PROGRAM F12_PackerQueuesCtrl
VAR

	rtrigScanBarcode				: R_TRIG;
	fbScannerCtrl					: FB_SCANNER_CameraSelect;
	fbImageBuffer					: FB_CASE_LastRowPoisitionBuffer_v2;
	fbCaseContentEvaluation			: FB_SCANNER_Evaluation;

	bShiftBufferDone						: BOOL;

	ctuAuxRowCounter				: CTU;
	nAuxRowIndex						: INT;
	rtrigAuxRowComplete				: R_TRIG;	(*option*)

	fbCaseInspectionSeq			: FB_SYSTEM_SeqControl;
	nSequenceStep				: INT;
	b00_Idle						: BOOL;
	b01_ScanBarcode				: BOOL;
	b06_MoveOutersToCaseData		: BOOL;
	b20_Done						: BOOL;

	bBusy						: BOOL;
	fbScanTimeout					: TON;

	fbFailedReadCounter			: CTU;
	fbMoveOuterToCaseDataPosition	: FB_CASE_MoveOutersRowToPacker;
	rtrigCaseContentValidation				: R_TRIG;

	fbValidationIndexOK						: FB_CTU32;
	fbValidationIndexUnder					: FB_CTU32;
	fbValidationIndexOver					: FB_CTU32;
	fbValidationNotFound					: FB_CTU32;

	tofCaseContentCameraOFFDelay 	: TOF;
	bTest	: BOOL;


	fbDebugCNT				: FB_DEBUG_CounterArray;
	aCNTDebug				: ARRAY [1..10] OF UDINT;
	bResetCNT					: BOOL;

END_VAR
(*
VAR CONSTANT
	sOptions						: ST_SCANNER_Options := (eScannerType := E_MV_420_FULL, nImageBuffer := 1, nExpectedResp := 1);
END_VAR*)

(*
Modification history:
Date		|	Author 		|	Remark
----------------------------------------------------------------------------------------------------
02.09.20	|	PP			|	Start Remarking.
*)
VAR // added by the converter: edge detectors and wires of the graphical bodies
    _w1 : BOOL;
END_VAR

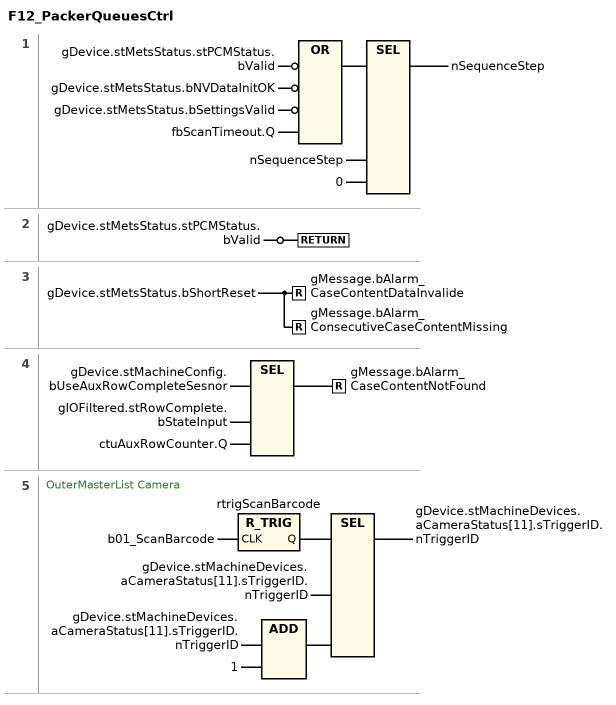
// NETWORK 1
nSequenceStep := SEL(NOT gDevice.stMetsStatus.stPCMStatus.bValid OR NOT gDevice.stMetsStatus.bNVDataInitOK OR NOT gDevice.stMetsStatus.bSettingsValid OR fbScanTimeout.Q, nSequenceStep, 0);

// NETWORK 2
IF NOT gDevice.stMetsStatus.stPCMStatus.bValid THEN RETURN; END_IF

// NETWORK 3
gMessage.bAlarm_CaseContentDataInvalide R= gDevice.stMetsStatus.bShortReset;
gMessage.bAlarm_ConsecutiveCaseContentMissing R= gDevice.stMetsStatus.bShortReset;

// NETWORK 4
gMessage.bAlarm_CaseContentNotFound R= SEL(gDevice.stMachineConfig.bUseAuxRowCompleteSesnor, gIOFiltered.stRowComplete.bStateInput, ctuAuxRowCounter.Q);

// NETWORK 5
// OuterMasterList Camera
rtrigScanBarcode(CLK := b01_ScanBarcode); // R_TRIG
gDevice.stMachineDevices.aCameraStatus[11].sTriggerID.nTriggerID := SEL(rtrigScanBarcode.Q, gDevice.stMachineDevices.aCameraStatus[11].sTriggerID.nTriggerID, gDevice.stMachineDevices.aCameraStatus[11].sTriggerID.nTriggerID + 1);

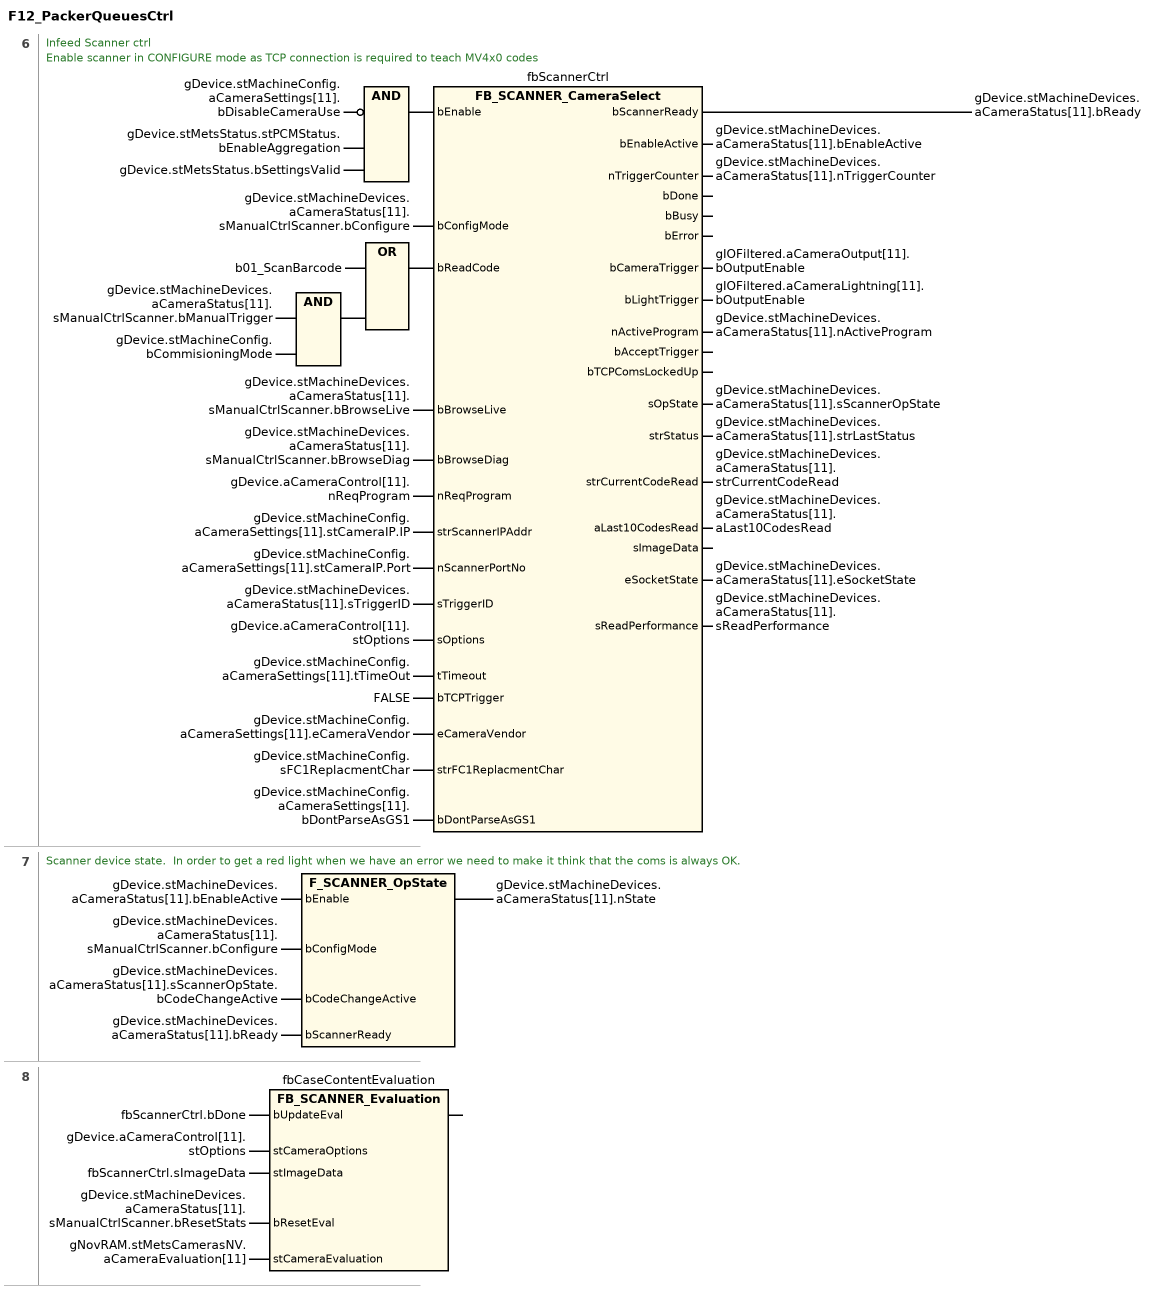
// NETWORK 6
// 					Infeed Scanner ctrl
// Enable scanner in CONFIGURE mode as TCP connection is required to teach MV4x0 codes
//
fbScannerCtrl(
    bEnable := NOT gDevice.stMachineConfig.aCameraSettings[11].bDisableCameraUse AND gDevice.stMetsStatus.stPCMStatus.bEnableAggregation AND gDevice.stMetsStatus.bSettingsValid,
    bConfigMode := gDevice.stMachineDevices.aCameraStatus[11].sManualCtrlScanner.bConfigure,
    bReadCode := b01_ScanBarcode OR gDevice.stMachineDevices.aCameraStatus[11].sManualCtrlScanner.bManualTrigger AND gDevice.stMachineConfig.bCommisioningMode,
    bBrowseLive := gDevice.stMachineDevices.aCameraStatus[11].sManualCtrlScanner.bBrowseLive,
    bBrowseDiag := gDevice.stMachineDevices.aCameraStatus[11].sManualCtrlScanner.bBrowseDiag,
    nReqProgram := gDevice.aCameraControl[11].nReqProgram,
    strScannerIPAddr := gDevice.stMachineConfig.aCameraSettings[11].stCameraIP.IP,
    nScannerPortNo := gDevice.stMachineConfig.aCameraSettings[11].stCameraIP.Port,
    sTriggerID := gDevice.stMachineDevices.aCameraStatus[11].sTriggerID,
    sOptions := gDevice.aCameraControl[11].stOptions,
    tTimeout := gDevice.stMachineConfig.aCameraSettings[11].tTimeOut,
    bTCPTrigger := FALSE,
    eCameraVendor := gDevice.stMachineConfig.aCameraSettings[11].eCameraVendor,
    strFC1ReplacmentChar := gDevice.stMachineConfig.sFC1ReplacmentChar,
    bDontParseAsGS1 := gDevice.stMachineConfig.aCameraSettings[11].bDontParseAsGS1,
    bEnableActive => gDevice.stMachineDevices.aCameraStatus[11].bEnableActive,
    nTriggerCounter => gDevice.stMachineDevices.aCameraStatus[11].nTriggerCounter,
    bCameraTrigger => gIOFiltered.aCameraOutput[11].bOutputEnable,
    bLightTrigger => gIOFiltered.aCameraLightning[11].bOutputEnable,
    nActiveProgram => gDevice.stMachineDevices.aCameraStatus[11].nActiveProgram,
    sOpState => gDevice.stMachineDevices.aCameraStatus[11].sScannerOpState,
    strStatus => gDevice.stMachineDevices.aCameraStatus[11].strLastStatus,
    strCurrentCodeRead => gDevice.stMachineDevices.aCameraStatus[11].strCurrentCodeRead,
    aLast10CodesRead => gDevice.stMachineDevices.aCameraStatus[11].aLast10CodesRead,
    eSocketState => gDevice.stMachineDevices.aCameraStatus[11].eSocketState,
    sReadPerformance => gDevice.stMachineDevices.aCameraStatus[11].sReadPerformance); // FB_SCANNER_CameraSelect
gDevice.stMachineDevices.aCameraStatus[11].bReady := fbScannerCtrl.bScannerReady;

// NETWORK 7
// Scanner device state.  In order to get a red light when we have an error we need to make it think that the coms is always OK.
gDevice.stMachineDevices.aCameraStatus[11].nState := F_SCANNER_OpState(bEnable := gDevice.stMachineDevices.aCameraStatus[11].bEnableActive, bConfigMode := gDevice.stMachineDevices.aCameraStatus[11].sManualCtrlScanner.bConfigure, bCodeChangeActive := gDevice.stMachineDevices.aCameraStatus[11].sScannerOpState.bCodeChangeActive, bScannerReady := gDevice.stMachineDevices.aCameraStatus[11].bReady);

// NETWORK 8
fbCaseContentEvaluation(
    bUpdateEval := fbScannerCtrl.bDone,
    stCameraOptions := gDevice.aCameraControl[11].stOptions,
    stImageData := fbScannerCtrl.sImageData,
    bResetEval := gDevice.stMachineDevices.aCameraStatus[11].sManualCtrlScanner.bResetStats,
    stCameraEvaluation := gNovRAM.stMetsCamerasNV.aCameraEvaluation[11]); // FB_SCANNER_Evaluation

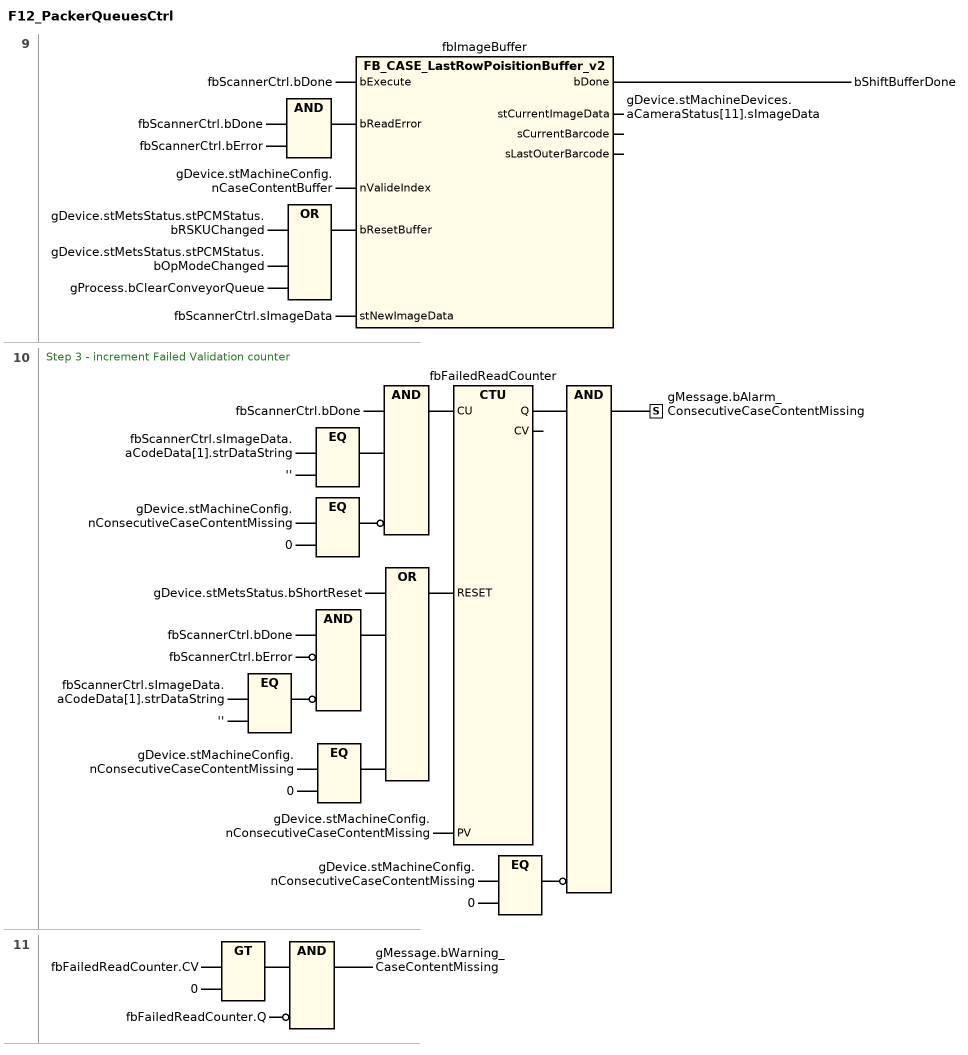
// NETWORK 9
fbImageBuffer(
    bExecute := fbScannerCtrl.bDone,
    bReadError := fbScannerCtrl.bDone AND fbScannerCtrl.bError,
    nValideIndex := gDevice.stMachineConfig.nCaseContentBuffer,
    bResetBuffer := gDevice.stMetsStatus.stPCMStatus.bRSKUChanged OR gDevice.stMetsStatus.stPCMStatus.bOpModeChanged OR gProcess.bClearConveyorQueue,
    stNewImageData := fbScannerCtrl.sImageData,
    stCurrentImageData => gDevice.stMachineDevices.aCameraStatus[11].sImageData); // FB_CASE_LastRowPoisitionBuffer_v2
bShiftBufferDone := fbImageBuffer.bDone;

// NETWORK 10
// Step 3 - increment Failed Validation counter
fbFailedReadCounter(
    CU := fbScannerCtrl.bDone AND fbScannerCtrl.sImageData.aCodeData[1].strDataString = '' AND NOT (gDevice.stMachineConfig.nConsecutiveCaseContentMissing = 0),
    RESET := gDevice.stMetsStatus.bShortReset OR fbScannerCtrl.bDone AND NOT fbScannerCtrl.bError AND NOT (fbScannerCtrl.sImageData.aCodeData[1].strDataString = '') OR gDevice.stMachineConfig.nConsecutiveCaseContentMissing = 0,
    PV := gDevice.stMachineConfig.nConsecutiveCaseContentMissing); // CTU
gMessage.bAlarm_ConsecutiveCaseContentMissing S= fbFailedReadCounter.Q AND NOT (gDevice.stMachineConfig.nConsecutiveCaseContentMissing = 0);

// NETWORK 11
gMessage.bWarning_CaseContentMissing := fbFailedReadCounter.CV > 0 AND NOT fbFailedReadCounter.Q;

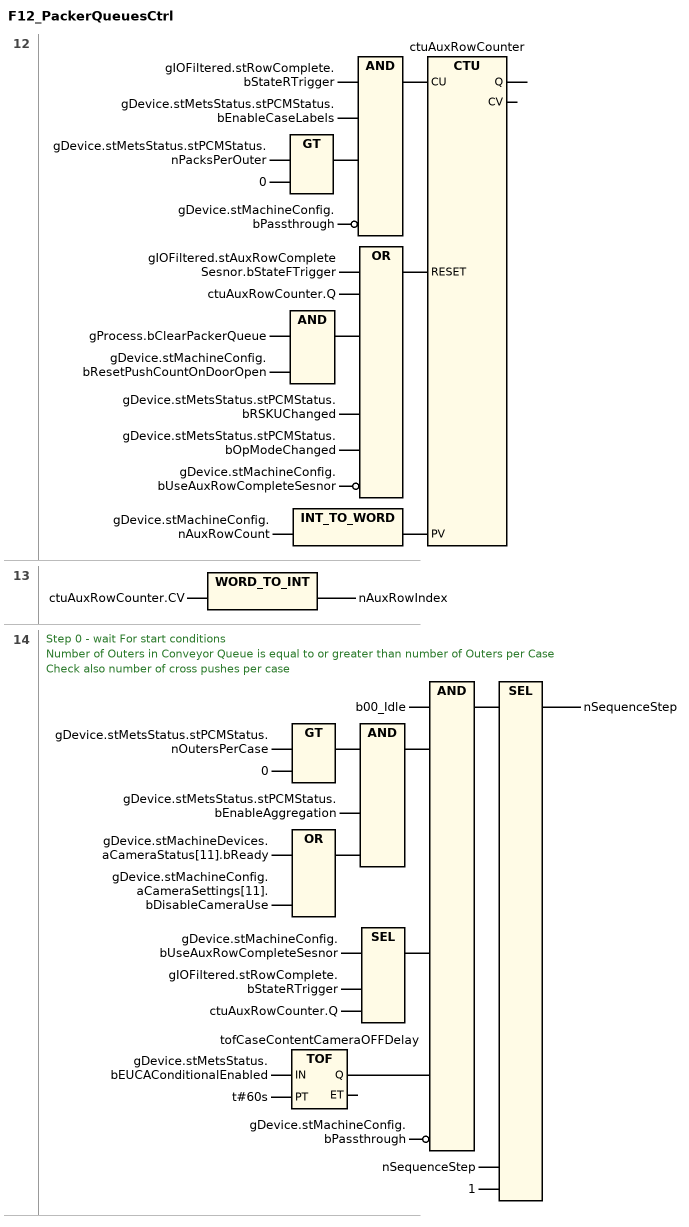
// NETWORK 12
ctuAuxRowCounter(
    CU := gIOFiltered.stRowComplete.bStateRTrigger AND gDevice.stMetsStatus.stPCMStatus.bEnableCaseLabels AND gDevice.stMetsStatus.stPCMStatus.nPacksPerOuter > 0 AND NOT gDevice.stMachineConfig.bPassthrough,
    RESET := gIOFiltered.stAuxRowCompleteSesnor.bStateFTrigger OR ctuAuxRowCounter.Q OR gProcess.bClearPackerQueue AND gDevice.stMachineConfig.bResetPushCountOnDoorOpen OR gDevice.stMetsStatus.stPCMStatus.bRSKUChanged OR gDevice.stMetsStatus.stPCMStatus.bOpModeChanged OR NOT gDevice.stMachineConfig.bUseAuxRowCompleteSesnor,
    PV := INT_TO_WORD(gDevice.stMachineConfig.nAuxRowCount)); // CTU

// NETWORK 13
nAuxRowIndex := WORD_TO_INT(ctuAuxRowCounter.CV);

// NETWORK 14
// 					Step 0 - wait For start conditions
// Number of Outers in Conveyor Queue is equal to or greater than number of Outers per Case
// Check also number of cross pushes per case
//
tofCaseContentCameraOFFDelay(IN := gDevice.stMetsStatus.bEUCAConditionalEnabled, PT := t#60s); // TOF
nSequenceStep := SEL(b00_Idle AND (gDevice.stMetsStatus.stPCMStatus.nOutersPerCase > 0 AND gDevice.stMetsStatus.stPCMStatus.bEnableAggregation AND (gDevice.stMachineDevices.aCameraStatus[11].bReady OR gDevice.stMachineConfig.aCameraSettings[11].bDisableCameraUse)) AND SEL(gDevice.stMachineConfig.bUseAuxRowCompleteSesnor, gIOFiltered.stRowComplete.bStateRTrigger, ctuAuxRowCounter.Q) AND tofCaseContentCameraOFFDelay.Q AND NOT gDevice.stMachineConfig.bPassthrough, nSequenceStep, 1);

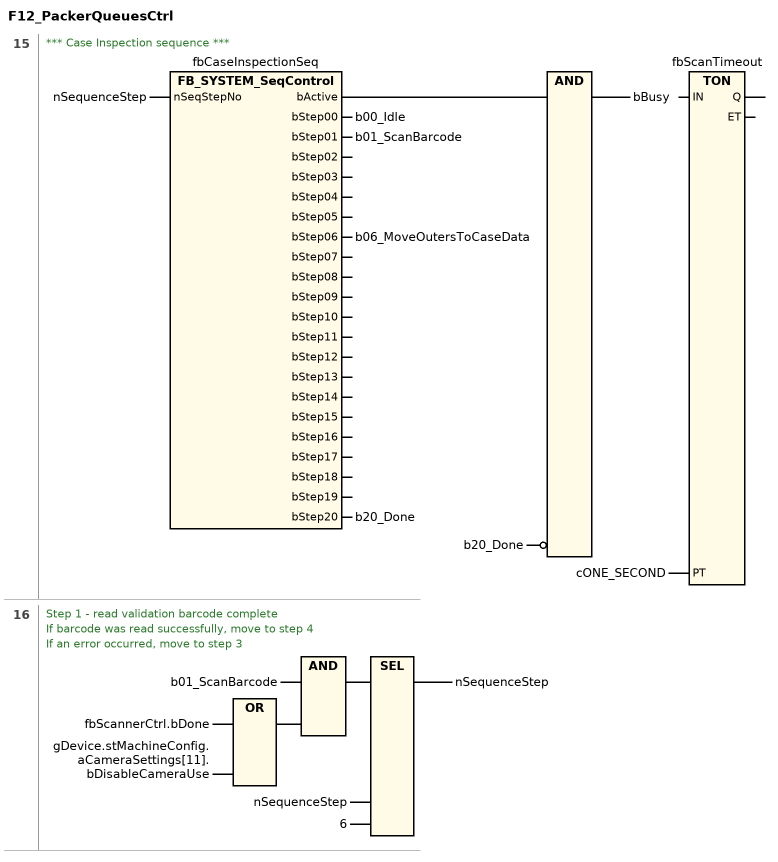
// NETWORK 15
// *** Case Inspection sequence ***
fbCaseInspectionSeq(
    nSeqStepNo := nSequenceStep,
    bStep00 => b00_Idle,
    bStep01 => b01_ScanBarcode,
    bStep06 => b06_MoveOutersToCaseData,
    bStep20 => b20_Done); // FB_SYSTEM_SeqControl
_w1 := fbCaseInspectionSeq.bActive AND NOT b20_Done;
bBusy := _w1;
fbScanTimeout(IN := _w1, PT := cONE_SECOND); // TON

// NETWORK 16
// 					Step 1 - read validation barcode complete
// If barcode was read successfully, move to step 4
// If an error occurred, move to step 3
//
nSequenceStep := SEL(b01_ScanBarcode AND (fbScannerCtrl.bDone OR gDevice.stMachineConfig.aCameraSettings[11].bDisableCameraUse), nSequenceStep, 6);

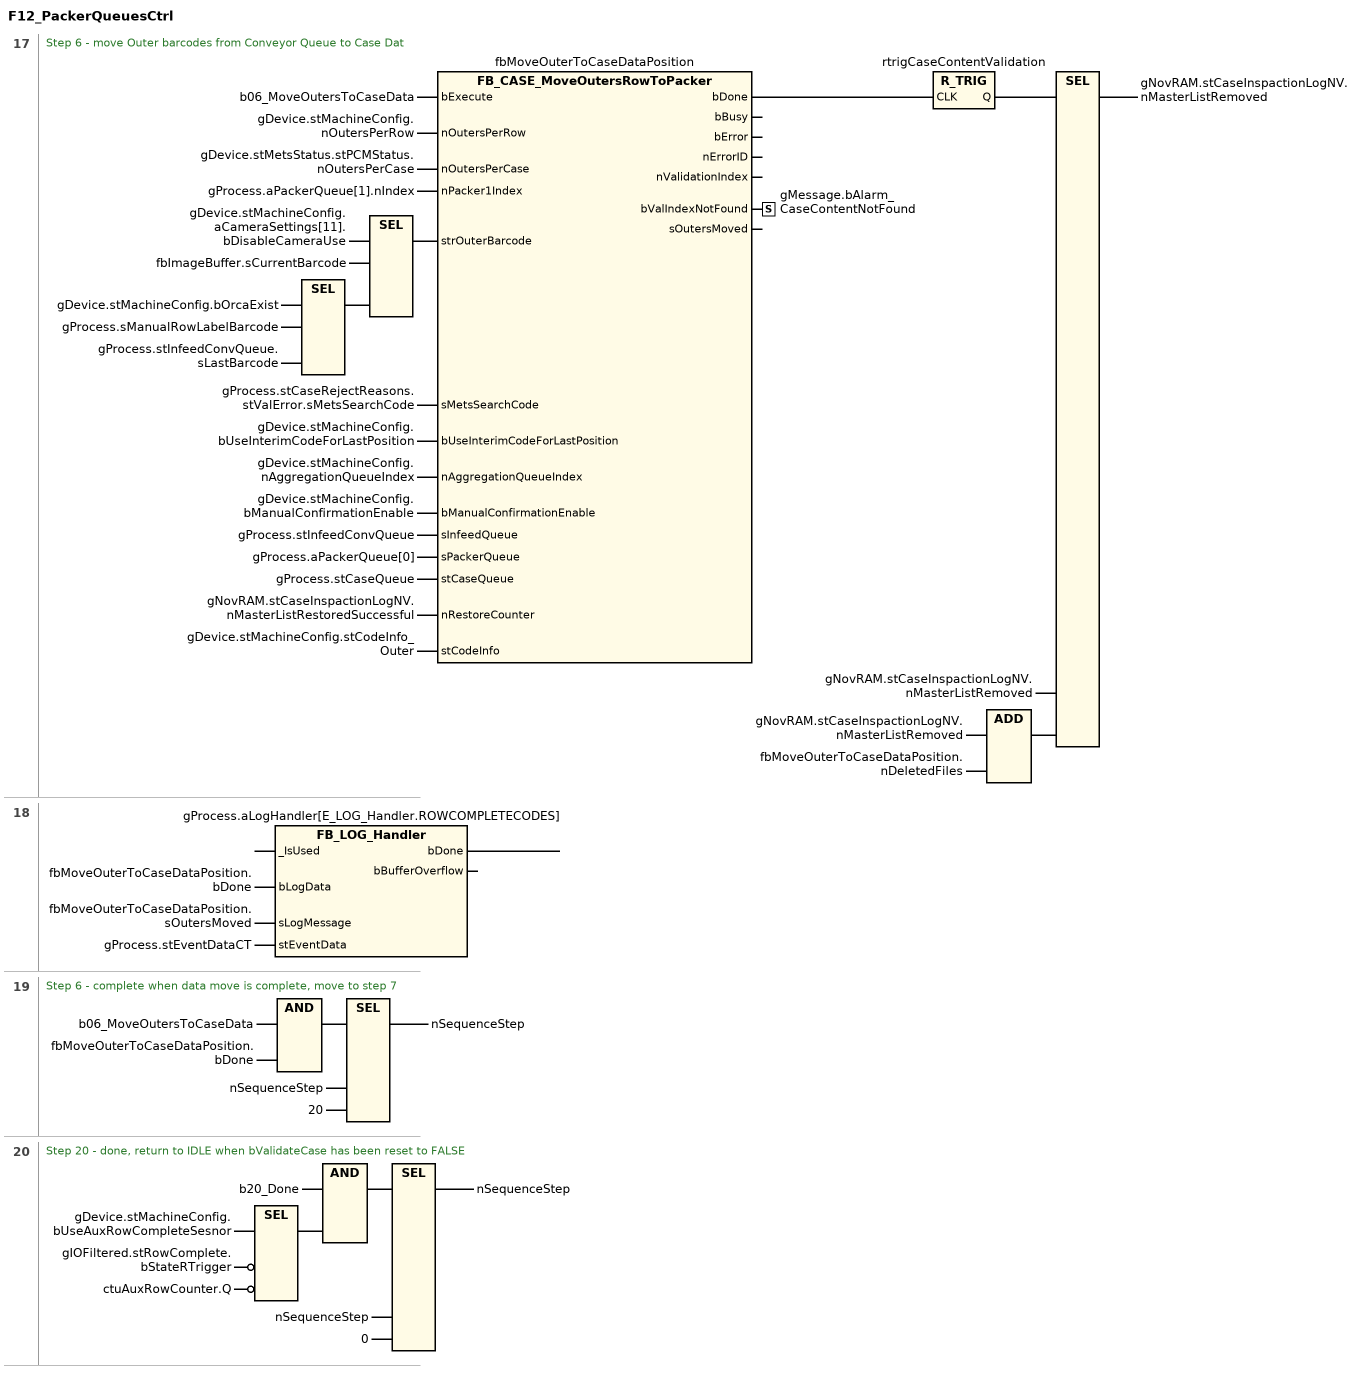
// NETWORK 17
// Step 6 - move Outer barcodes from Conveyor Queue to Case Dat
fbMoveOuterToCaseDataPosition(
    bExecute := b06_MoveOutersToCaseData,
    nOutersPerRow := gDevice.stMachineConfig.nOutersPerRow,
    nOutersPerCase := gDevice.stMetsStatus.stPCMStatus.nOutersPerCase,
    nPacker1Index := gProcess.aPackerQueue[1].nIndex,
    strOuterBarcode := SEL(gDevice.stMachineConfig.aCameraSettings[11].bDisableCameraUse, fbImageBuffer.sCurrentBarcode, SEL(gDevice.stMachineConfig.bOrcaExist, gProcess.sManualRowLabelBarcode, gProcess.stInfeedConvQueue.sLastBarcode)),
    sMetsSearchCode := gProcess.stCaseRejectReasons.stValError.sMetsSearchCode,
    bUseInterimCodeForLastPosition := gDevice.stMachineConfig.bUseInterimCodeForLastPosition,
    nAggregationQueueIndex := gDevice.stMachineConfig.nAggregationQueueIndex,
    bManualConfirmationEnable := gDevice.stMachineConfig.bManualConfirmationEnable,
    sInfeedQueue := gProcess.stInfeedConvQueue,
    sPackerQueue := gProcess.aPackerQueue[0],
    stCaseQueue := gProcess.stCaseQueue,
    nRestoreCounter := gNovRAM.stCaseInspactionLogNV.nMasterListRestoredSuccessful,
    stCodeInfo := gDevice.stMachineConfig.stCodeInfo_Outer); // FB_CASE_MoveOutersRowToPacker
gMessage.bAlarm_CaseContentNotFound S= fbMoveOuterToCaseDataPosition.bValIndexNotFound;
rtrigCaseContentValidation(CLK := fbMoveOuterToCaseDataPosition.bDone); // R_TRIG
gNovRAM.stCaseInspactionLogNV.nMasterListRemoved := SEL(rtrigCaseContentValidation.Q, gNovRAM.stCaseInspactionLogNV.nMasterListRemoved, gNovRAM.stCaseInspactionLogNV.nMasterListRemoved + fbMoveOuterToCaseDataPosition.nDeletedFiles);

// NETWORK 18
gProcess.aLogHandler[E_LOG_Handler.ROWCOMPLETECODES](
    bLogData := fbMoveOuterToCaseDataPosition.bDone,
    sLogMessage := fbMoveOuterToCaseDataPosition.sOutersMoved,
    stEventData := gProcess.stEventDataCT); // FB_LOG_Handler

// NETWORK 19
// Step 6 - complete when data move is complete, move to step 7
nSequenceStep := SEL(b06_MoveOutersToCaseData AND fbMoveOuterToCaseDataPosition.bDone, nSequenceStep, 20);

// NETWORK 20
// Step 20 - done, return to IDLE when bValidateCase has been reset to FALSE
nSequenceStep := SEL(b20_Done AND SEL(gDevice.stMachineConfig.bUseAuxRowCompleteSesnor, NOT gIOFiltered.stRowComplete.bStateRTrigger, NOT ctuAuxRowCounter.Q), nSequenceStep, 0);

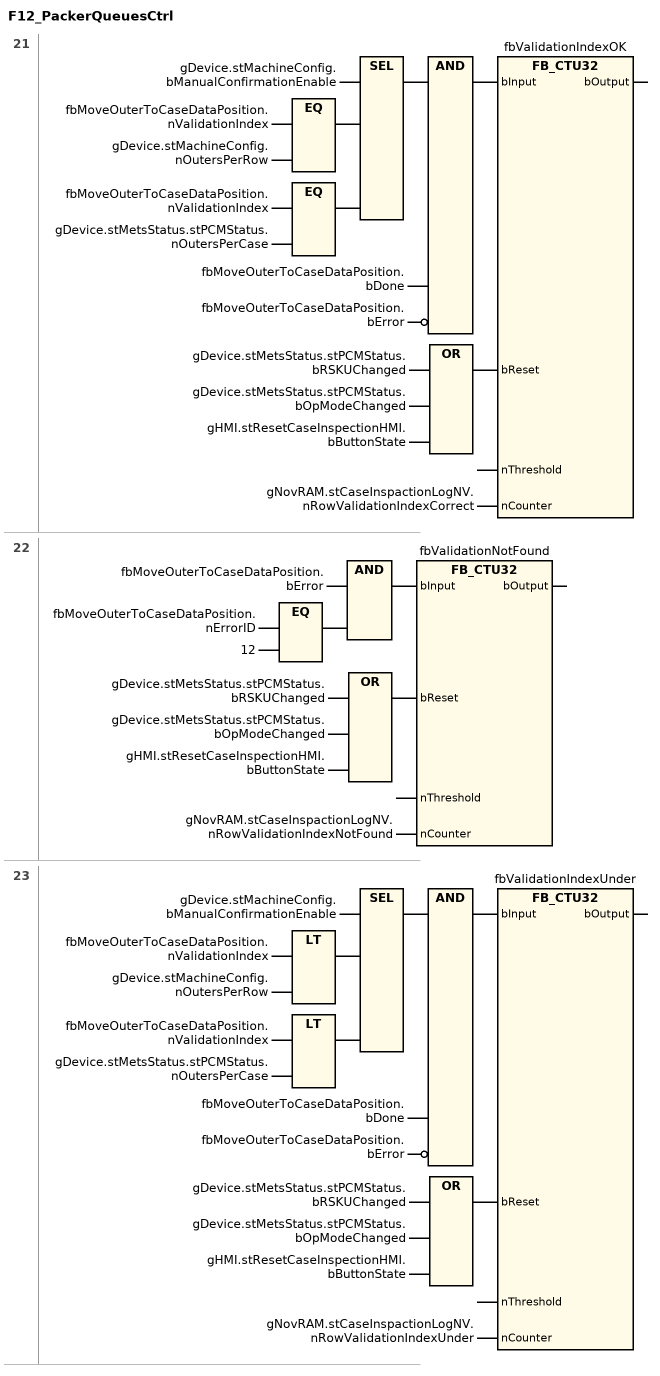
// NETWORK 21
fbValidationIndexOK(
    bInput := SEL(gDevice.stMachineConfig.bManualConfirmationEnable, fbMoveOuterToCaseDataPosition.nValidationIndex = gDevice.stMachineConfig.nOutersPerRow, fbMoveOuterToCaseDataPosition.nValidationIndex = gDevice.stMetsStatus.stPCMStatus.nOutersPerCase) AND fbMoveOuterToCaseDataPosition.bDone AND NOT fbMoveOuterToCaseDataPosition.bError,
    bReset := gDevice.stMetsStatus.stPCMStatus.bRSKUChanged OR gDevice.stMetsStatus.stPCMStatus.bOpModeChanged OR gHMI.stResetCaseInspectionHMI.bButtonState,
    nCounter := gNovRAM.stCaseInspactionLogNV.nRowValidationIndexCorrect); // FB_CTU32

// NETWORK 22
fbValidationNotFound(
    bInput := fbMoveOuterToCaseDataPosition.bError AND fbMoveOuterToCaseDataPosition.nErrorID = 12,
    bReset := gDevice.stMetsStatus.stPCMStatus.bRSKUChanged OR gDevice.stMetsStatus.stPCMStatus.bOpModeChanged OR gHMI.stResetCaseInspectionHMI.bButtonState,
    nCounter := gNovRAM.stCaseInspactionLogNV.nRowValidationIndexNotFound); // FB_CTU32

// NETWORK 23
fbValidationIndexUnder(
    bInput := SEL(gDevice.stMachineConfig.bManualConfirmationEnable, fbMoveOuterToCaseDataPosition.nValidationIndex < gDevice.stMachineConfig.nOutersPerRow, fbMoveOuterToCaseDataPosition.nValidationIndex < gDevice.stMetsStatus.stPCMStatus.nOutersPerCase) AND fbMoveOuterToCaseDataPosition.bDone AND NOT fbMoveOuterToCaseDataPosition.bError,
    bReset := gDevice.stMetsStatus.stPCMStatus.bRSKUChanged OR gDevice.stMetsStatus.stPCMStatus.bOpModeChanged OR gHMI.stResetCaseInspectionHMI.bButtonState,
    nCounter := gNovRAM.stCaseInspactionLogNV.nRowValidationIndexUnder); // FB_CTU32

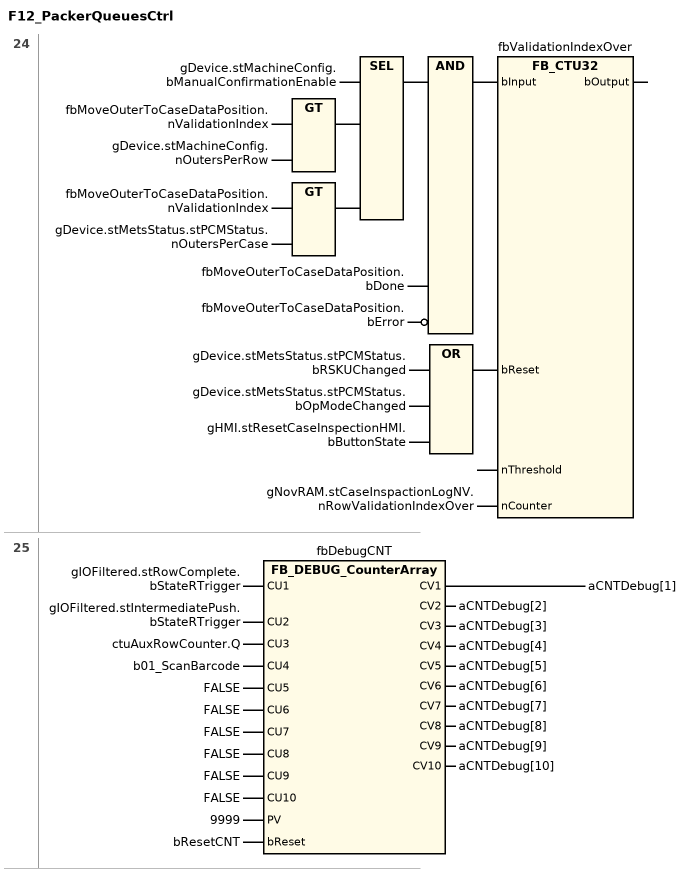
// NETWORK 24
fbValidationIndexOver(
    bInput := SEL(gDevice.stMachineConfig.bManualConfirmationEnable, fbMoveOuterToCaseDataPosition.nValidationIndex > gDevice.stMachineConfig.nOutersPerRow, fbMoveOuterToCaseDataPosition.nValidationIndex > gDevice.stMetsStatus.stPCMStatus.nOutersPerCase) AND fbMoveOuterToCaseDataPosition.bDone AND NOT fbMoveOuterToCaseDataPosition.bError,
    bReset := gDevice.stMetsStatus.stPCMStatus.bRSKUChanged OR gDevice.stMetsStatus.stPCMStatus.bOpModeChanged OR gHMI.stResetCaseInspectionHMI.bButtonState,
    nCounter := gNovRAM.stCaseInspactionLogNV.nRowValidationIndexOver); // FB_CTU32

// NETWORK 25
fbDebugCNT(
    CU1 := gIOFiltered.stRowComplete.bStateRTrigger,
    CU2 := gIOFiltered.stIntermediatePush.bStateRTrigger,
    CU3 := ctuAuxRowCounter.Q,
    CU4 := b01_ScanBarcode,
    CU5 := FALSE,
    CU6 := FALSE,
    CU7 := FALSE,
    CU8 := FALSE,
    CU9 := FALSE,
    CU10 := FALSE,
    PV := 9999,
    bReset := bResetCNT,
    CV2 => aCNTDebug[2],
    CV3 => aCNTDebug[3],
    CV4 => aCNTDebug[4],
    CV5 => aCNTDebug[5],
    CV6 => aCNTDebug[6],
    CV7 => aCNTDebug[7],
    CV8 => aCNTDebug[8],
    CV9 => aCNTDebug[9],
    CV10 => aCNTDebug[10]); // FB_DEBUG_CounterArray
aCNTDebug[1] := fbDebugCNT.CV1;

END_PROGRAM

(* stored: Version 1.1.0.1
   POU F12_PackerQueuesCtrl: Id {a3a5fe0e-de1b-4002-8715-78c18abb42e0}, SpecialFunc None *)
